// TIA Portal V17 export
// export: Created 2025-06-26T07:49:15.3726459Z, ExportSetting WithDefaults, DisplayName Totally Integrated Automation Portal, DisplayVersion V17 Update 8, DisplayName TIA Portal Openness, DisplayVersion V17 Update 8, DisplayName TIA Portal Version Control Interface, DisplayVersion V17, DisplayName STEP 7 Professional, DisplayVersion V17 Update 8, DisplayName STEP 7 Safety, DisplayVersion V17 Update 6, DisplayName WinCC Advanced, DisplayVersion V17 Update 8
FUNCTION_BLOCK "Customer"   // FB3, LAD
TITLE = Combine signals from Customer into DB_Application
{ S7_Optimized_Access := 'TRUE' }
AUTHOR : Heaten
VERSION : 0.1
// stored: AutoNumber true, IsIECCheckEnabled false, IsRetainMemResEnabled false, MemoryReserve 100, SetENOAutomatically false, UDAEnableTagReadback false
   VAR
      Watchdog { S7_SetPoint := 'True'} : "fbHeartbeatCount2";
      epStartRequest { S7_SetPoint := 'True'} : Bool;
      enStartRequest : Bool;
      epStopRequest : Bool;
      enStopRequest : Bool;
      epAlarmAcknowledge : Bool;
      enAlarmAcknowledge : Bool;
      epResetEmergencyStop : Bool;
      enResetEmergencyStop : Bool;
      SetpointPrev : Real;
      RegulationTargetPrev : Int;
      HCV812Cmd : Real;   // TEMPORARY
      HCV815Cmd : Real;   // TEMPORARY
      HCV818Cmd : Real;   // TEMPORARY
      HCV821Cmd : Real;   // TEMPORARY
   END_VAR
   VAR_TEMP
      bWatchdogOk : Bool;
      bStopReq : Bool;
      fDummy : Real;
      iDummy : Int;
   END_VAR
   VAR_TEMP   // added for the SCL form of the ladder/FBD networks
      _w1 : Bool;
      _w2 : Bool;
      _w3 : Bool;
      _w4 : Bool;
   END_VAR
BEGIN

REGION Network 1: Map IO tags to DBs
   // When using S7 communication this mapping is not necessary
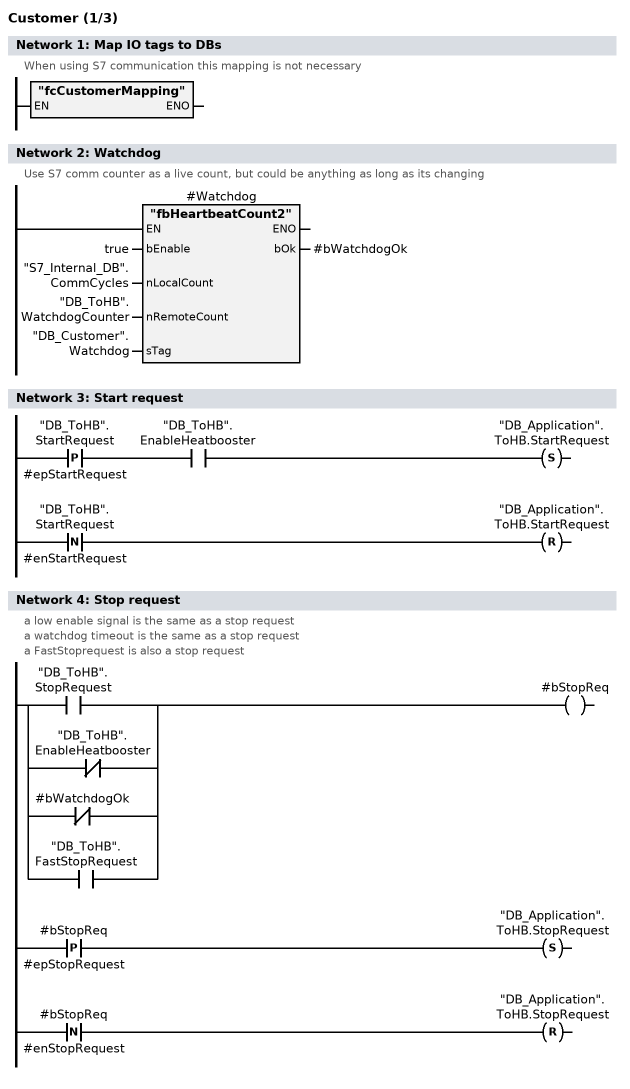
   RUNG wire#powerrail
      "fcCustomerMapping"()
   END_RUNG
   // the same network as SCL:
   "fcCustomerMapping"();
END_REGION

REGION Network 2: Watchdog
   // Use S7 comm counter as a live count, but could be anything as long as its changing
   RUNG wire#powerrail
      #Watchdog(bEnable := true, nLocalCount := "S7_Internal_DB".CommCycles, nRemoteCount := "DB_ToHB".WatchdogCounter, sTag := "DB_Customer".Watchdog, bOk => #bWatchdogOk)
   END_RUNG
   // the same network as SCL:
   #Watchdog(bEnable := true,   // "fbHeartbeatCount2"
             nLocalCount := "S7_Internal_DB".CommCycles,
             nRemoteCount := "DB_ToHB".WatchdogCounter,
             sTag := "DB_Customer".Watchdog,
             bOk => #bWatchdogOk);
END_REGION

REGION Network 3: Start request
   RUNG wire#powerrail
      P_Contact(operand := "DB_ToHB".StartRequest, bit := #epStartRequest)
      Contact( "DB_ToHB".EnableHeatbooster )
      S_Coil( "DB_Application".ToHB.StartRequest )
   END_RUNG
   RUNG wire#powerrail
      N_Contact(operand := "DB_ToHB".StartRequest, bit := #enStartRequest)
      R_Coil( "DB_Application".ToHB.StartRequest )
   END_RUNG
   // the same network as SCL:
   #_w1 := "DB_ToHB".StartRequest AND NOT #epStartRequest;   // rising edge of "DB_ToHB".StartRequest
   #epStartRequest := "DB_ToHB".StartRequest;
   IF #_w1 AND "DB_ToHB".EnableHeatbooster THEN "DB_Application".ToHB.StartRequest := TRUE; END_IF;
   #_w2 := NOT "DB_ToHB".StartRequest AND #enStartRequest;   // falling edge of "DB_ToHB".StartRequest
   #enStartRequest := "DB_ToHB".StartRequest;
   IF #_w2 THEN "DB_Application".ToHB.StartRequest := FALSE; END_IF;
END_REGION

REGION Network 4: Stop request
   // a low enable signal is the same as a stop request
   // a watchdog timeout is the same as a stop request
   // a FastStoprequest is also a stop request
   RUNG wire#powerrail
      Contact( "DB_ToHB".StopRequest )
      wire#w1
      Coil( #bStopReq )
   END_RUNG
   RUNG wire#powerrail
      I_Contact( "DB_ToHB".EnableHeatbooster )
   END_RUNG wire#w1
   RUNG wire#powerrail
      I_Contact( #bWatchdogOk )
   END_RUNG wire#w1
   RUNG wire#powerrail
      Contact( "DB_ToHB".FastStopRequest )
   END_RUNG wire#w1
   RUNG wire#powerrail
      P_Contact(operand := #bStopReq, bit := #epStopRequest)
      S_Coil( "DB_Application".ToHB.StopRequest )
   END_RUNG
   RUNG wire#powerrail
      N_Contact(operand := #bStopReq, bit := #enStopRequest)
      R_Coil( "DB_Application".ToHB.StopRequest )
   END_RUNG
   // the same network as SCL:
   #bStopReq := "DB_ToHB".StopRequest OR NOT "DB_ToHB".EnableHeatbooster OR NOT #bWatchdogOk OR "DB_ToHB".FastStopRequest;
   #_w1 := #bStopReq AND NOT #epStopRequest;   // rising edge of #bStopReq
   #epStopRequest := #bStopReq;
   IF #_w1 THEN "DB_Application".ToHB.StopRequest := TRUE; END_IF;
   #_w2 := NOT #bStopReq AND #enStopRequest;   // falling edge of #bStopReq
   #enStopRequest := #bStopReq;
   IF #_w2 THEN "DB_Application".ToHB.StopRequest := FALSE; END_IF;
END_REGION

REGION Network 5: Commands
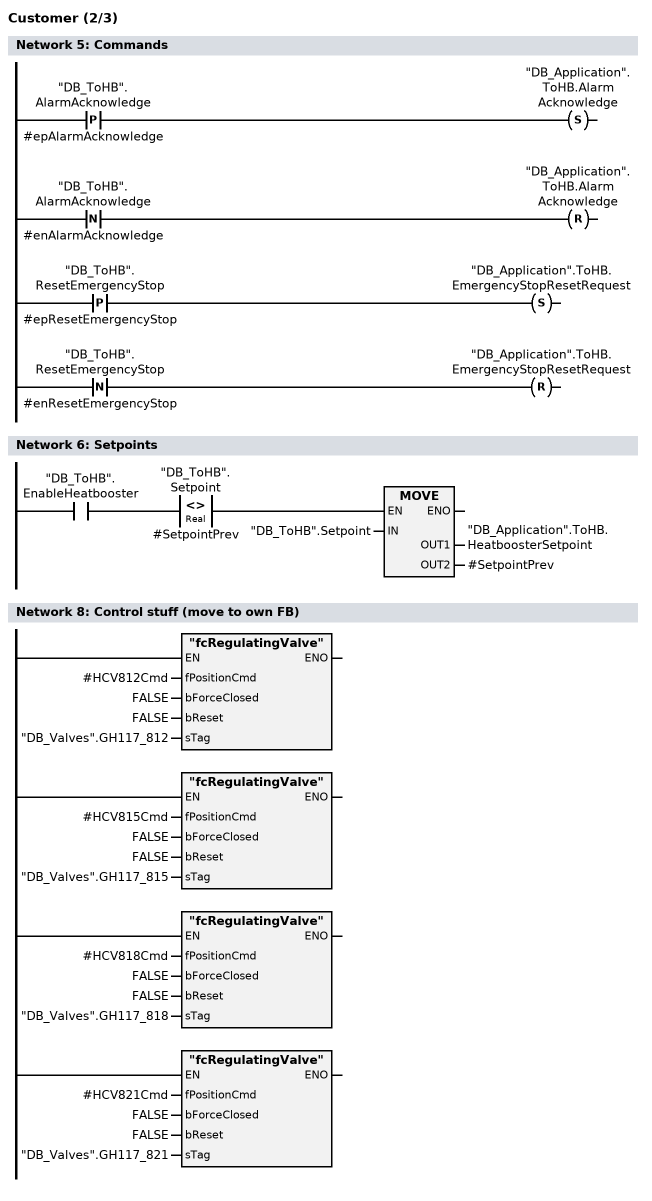
   RUNG wire#powerrail
      P_Contact(operand := "DB_ToHB".AlarmAcknowledge, bit := #epAlarmAcknowledge)
      S_Coil( "DB_Application".ToHB.AlarmAcknowledge )
   END_RUNG
   RUNG wire#powerrail
      N_Contact(operand := "DB_ToHB".AlarmAcknowledge, bit := #enAlarmAcknowledge)
      R_Coil( "DB_Application".ToHB.AlarmAcknowledge )
   END_RUNG
   RUNG wire#powerrail
      P_Contact(operand := "DB_ToHB".ResetEmergencyStop, bit := #epResetEmergencyStop)
      S_Coil( "DB_Application".ToHB.EmergencyStopResetRequest )
   END_RUNG
   RUNG wire#powerrail
      N_Contact(operand := "DB_ToHB".ResetEmergencyStop, bit := #enResetEmergencyStop)
      R_Coil( "DB_Application".ToHB.EmergencyStopResetRequest )
   END_RUNG
   // the same network as SCL:
   #_w1 := "DB_ToHB".AlarmAcknowledge AND NOT #epAlarmAcknowledge;   // rising edge of "DB_ToHB".AlarmAcknowledge
   #epAlarmAcknowledge := "DB_ToHB".AlarmAcknowledge;
   IF #_w1 THEN "DB_Application".ToHB.AlarmAcknowledge := TRUE; END_IF;
   #_w2 := NOT "DB_ToHB".AlarmAcknowledge AND #enAlarmAcknowledge;   // falling edge of "DB_ToHB".AlarmAcknowledge
   #enAlarmAcknowledge := "DB_ToHB".AlarmAcknowledge;
   IF #_w2 THEN "DB_Application".ToHB.AlarmAcknowledge := FALSE; END_IF;
   #_w3 := "DB_ToHB".ResetEmergencyStop AND NOT #epResetEmergencyStop;   // rising edge of "DB_ToHB".ResetEmergencyStop
   #epResetEmergencyStop := "DB_ToHB".ResetEmergencyStop;
   IF #_w3 THEN "DB_Application".ToHB.EmergencyStopResetRequest := TRUE; END_IF;
   #_w4 := NOT "DB_ToHB".ResetEmergencyStop AND #enResetEmergencyStop;   // falling edge of "DB_ToHB".ResetEmergencyStop
   #enResetEmergencyStop := "DB_ToHB".ResetEmergencyStop;
   IF #_w4 THEN "DB_Application".ToHB.EmergencyStopResetRequest := FALSE; END_IF;
END_REGION

REGION Network 6: Setpoints
   RUNG wire#powerrail
      Contact( "DB_ToHB".EnableHeatbooster )
      { S7_Templates := "SrcType := Real" } NE_Contact(in1 := "DB_ToHB".Setpoint, in2 := #SetpointPrev)
      Move(in := "DB_ToHB".Setpoint, out1 => "DB_Application".ToHB.HeatboosterSetpoint, out2 => #SetpointPrev)
   END_RUNG
   // the same network as SCL:
   IF "DB_ToHB".EnableHeatbooster AND ("DB_ToHB".Setpoint <> #SetpointPrev) THEN
       "DB_Application".ToHB.HeatboosterSetpoint := "DB_ToHB".Setpoint;
       #SetpointPrev := "DB_ToHB".Setpoint;
   END_IF;
END_REGION

REGION Network 7 (SCL): To Customer
   "DB_FromHB".CompressorMotorPower            := "DB_Heatbooster".Inverter.HBL_SC_10_A3.fValue;
   "DB_FromHB".CompressorMotorSpeed            := "DB_Heatbooster".Inverter.HBL_SC_10_A1.fValue;
   //"DB_FromHB".HBL_CT_524                      := "DB_Heatbooster".AI.HBL_CT_524.fValue;
   //"DB_FromHB".HBL_CT_538                      := "DB_Heatbooster".AI.HBL_CT_538.fValue;
   "DB_FromHB".HBL_CT_615    := "DB_Heatbooster".AI.HBL_TT_546.fValue;
   "DB_FromHB".HBL_CT_620  := "DB_Heatbooster".AI.HBL_TT_542.fValue;
   "DB_FromHB".HBL_SC_02_A3         := "DB_Heatbooster".AI.HBL_TT_16.fValue;
   "DB_FromHB".HBL_SC_10_A1    := "DB_Heatbooster".AI.HBL_TT_17.fValue;
   "DB_FromHB".HBL_SC_10_A2           := "DB_Heatbooster".AI.HBL_TT_18.fValue;

   "DB_FromHB".HBL_CT_643   := "DB_Heatbooster".AI.HBL_CT_01.fValue;
   "DB_FromHB".HBL_CT_673 := "DB_Heatbooster".AI.HBL_CT_615.fValue;
   "DB_FromHB".HBL_CT_950 := "DB_Heatbooster".AI.HBL_CT_03.fValue;
   "DB_FromHB".HBL_SC_10_A3 := "DB_Heatbooster".AI.SSC_LT_01.fValue;
   "DB_FromHB".TemperatureLift                 := "DB_Heatbooster".Calc.System.TemperatureLift.fValue;
   "DB_FromHB".COP                             := "DB_Heatbooster".Calc.System.COP.fValue;
   "DB_FromHB".HeatSinkHeatRate                := "DB_Heatbooster".Calc.HeatSink.HeatRate.fValue;
   "DB_FromHB".CompressorMotorPower := "DB_Heatbooster".Calc.System.ElectricalPower.fValue;
   "DB_FromHB".HeatboosterPerformance             := "DB_Application".FromHB.HeatboosterSetpoint;
   //"DB_FromHB".WatchdogCounter                := "DB_Application".FromHB.RegulationTarget;
   "DB_FromHB".RunningTimeHours                := INT_TO_UINT("DB_Application".FromHB.RunningTimeHours);
   "DB_FromHB".RunningTimeMinutes              := "DB_Application".FromHB.RunningTimeMinutes;
   "DB_FromHB".RunningTimeSeconds              := "DB_Application".FromHB.RunningTimeSeconds;

   "DB_FromHB".HeatboosterState                := "DB_Application".FromHB.MachineState;
   "DB_FromHB".EmergencyStopStatus             := "DB_Application".FromHB.EmergencyStop;
   "DB_FromHB".HBL_EC_01 := "DB_DO".HBL_EC_01;
   "DB_FromHB".HBL_EC_02 := "DB_DO".HBL_EC_02;
   "DB_FromHB".AlarmActive                    := "DB_DO".GH117_826_1;
   "DB_FromHB".WarningActive                    := "DB_DO".GH117_826_2;

   "DB_FromHB".Alarms                          := "DB_Application".FromHB.Alarms;
   //"DB_FromHB".HBL_SC_03_A1 := FALSE;
   //"DB_FromHB".HBL_SC_03_A2:= FALSE;
   //"DB_FromHB".HBL_SC_03_A3   := FALSE;
   //"DB_FromHB".HBL_SC_01_A1  := FALSE;
   //"DB_FromHB".HBL_SC_01_A2          := 0.0;
   "DB_FromHB".HBL_SC_01_A3            := 0.0;
   "DB_FromHB".HBL_SC_02_A1            := 0.0;
   "DB_FromHB".HBL_SC_02_A2              := 0.0;
   "DB_FromHB".WatchdogCounter                 := "DB_Customer".Watchdog.nLocalCount;
END_REGION

REGION Network 8: Control stuff (move to own FB)
   RUNG wire#powerrail
      "fcRegulatingValve"(fPositionCmd := #HCV812Cmd, bForceClosed := FALSE, bReset := FALSE, sTag := "DB_Valves".GH117_812)
   END_RUNG
   RUNG wire#powerrail
      "fcRegulatingValve"(fPositionCmd := #HCV815Cmd, bForceClosed := FALSE, bReset := FALSE, sTag := "DB_Valves".GH117_815)
   END_RUNG
   RUNG wire#powerrail
      "fcRegulatingValve"(fPositionCmd := #HCV818Cmd, bForceClosed := FALSE, bReset := FALSE, sTag := "DB_Valves".GH117_818)
   END_RUNG
   RUNG wire#powerrail
      "fcRegulatingValve"(fPositionCmd := #HCV821Cmd, bForceClosed := FALSE, bReset := FALSE, sTag := "DB_Valves".GH117_821)
   END_RUNG
   // the same network as SCL:
   "fcRegulatingValve"(fPositionCmd := #HCV812Cmd,
                       bForceClosed := FALSE,
                       bReset := FALSE,
                       sTag := "DB_Valves".GH117_812);
   "fcRegulatingValve"(fPositionCmd := #HCV815Cmd,
                       bForceClosed := FALSE,
                       bReset := FALSE,
                       sTag := "DB_Valves".GH117_815);
   "fcRegulatingValve"(fPositionCmd := #HCV818Cmd,
                       bForceClosed := FALSE,
                       bReset := FALSE,
                       sTag := "DB_Valves".GH117_818);
   "fcRegulatingValve"(fPositionCmd := #HCV821Cmd,
                       bForceClosed := FALSE,
                       bReset := FALSE,
                       sTag := "DB_Valves".GH117_821);
END_REGION

REGION Network 9: Analog outputs
   // Move to own FB in Section 30
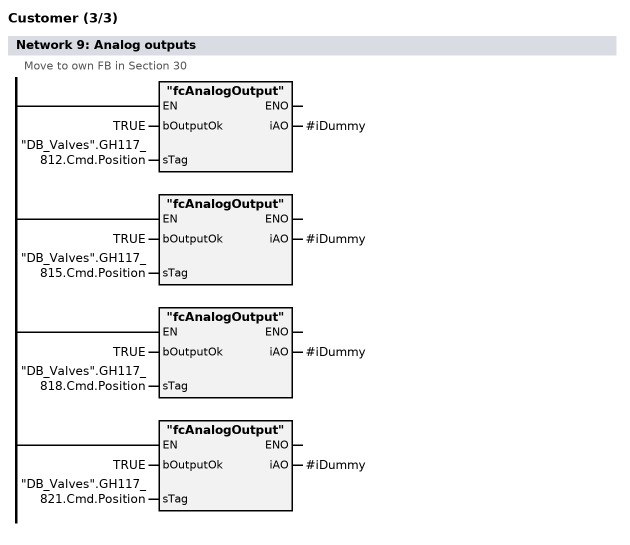
   RUNG wire#powerrail
      "fcAnalogOutput"(bOutputOk := TRUE, sTag := "DB_Valves".GH117_812.Cmd.Position, iAO => #iDummy)
   END_RUNG
   RUNG wire#powerrail
      "fcAnalogOutput"(bOutputOk := TRUE, sTag := "DB_Valves".GH117_815.Cmd.Position, iAO => #iDummy)
   END_RUNG
   RUNG wire#powerrail
      "fcAnalogOutput"(bOutputOk := TRUE, sTag := "DB_Valves".GH117_818.Cmd.Position, iAO => #iDummy)
   END_RUNG
   RUNG wire#powerrail
      "fcAnalogOutput"(bOutputOk := TRUE, sTag := "DB_Valves".GH117_821.Cmd.Position, iAO => #iDummy)
   END_RUNG
   // the same network as SCL:
   "fcAnalogOutput"(bOutputOk := TRUE, sTag := "DB_Valves".GH117_812.Cmd.Position, iAO => #iDummy);
   "fcAnalogOutput"(bOutputOk := TRUE, sTag := "DB_Valves".GH117_815.Cmd.Position, iAO => #iDummy);
   "fcAnalogOutput"(bOutputOk := TRUE, sTag := "DB_Valves".GH117_818.Cmd.Position, iAO => #iDummy);
   "fcAnalogOutput"(bOutputOk := TRUE, sTag := "DB_Valves".GH117_821.Cmd.Position, iAO => #iDummy);
END_REGION
END_FUNCTION_BLOCK
